INTERFACE I_DS402DriveCommon

END_INTERFACE

(* stored: Version 1.1.0.1
   Itf I_DS402DriveCommon: Id {5cfa6b6b-bfba-4af4-97dd-dc8ae67741ad} *)
